(* IEC 61131-3 sources: ahu-codesys/codesys/src/04-smoke-safety, 2 files *)

(* ---- GVL_Smoke.st ---- *)
{attribute 'qualified_only'}
VAR_GLOBAL
	(* Inputs *)
	SmokeDetected : BOOL;
	ResetSmoke : BOOL;

	(* Internal *)
	SmokeAlarmMem : BOOL;

	(* Outputs *)
	SmokeAlarm : BOOL;
END_VAR

(* ---- PLC_PRG_Smoke.st ---- *)
(* ======================
   Smoke Safety Interlock
   ====================== *)
(* Because safety takes priority over process control, smoke alarm must override motor and heating inputs *)

(* Smoke alarm latch - stays active until manually reset *)
GVL_Smoke.SmokeAlarmMem := (GVL_Smoke.SmokeDetected OR GVL_Smoke.SmokeAlarmMem) AND NOT GVL_Smoke.ResetSmoke;

(* Smoke Alarm Output *)
GVL_Smoke.SmokeAlarm := GVL_Smoke.SmokeAlarmMem;

(* Safety override - shut down all outputs on smoke alarm *)
(* This modifies outputs set by earlier logic sections *)

IF GVL_Smoke.SmokeAlarmMem THEN
	GVL.MotorInternal := FALSE;
	GVL.MotorOut := FALSE;
	GVL_Temp.HeatOutput := FALSE;
END_IF
